Universal Robots PolyScope program: TEST_SUB_109.urp

Program TEST_SUB_109 (installation=GD directory=/programs/GD createdIn=5.13.0 lastSavedIn=5.13.0 robotSerialNumber=20235201009)
Calibrated DH parameters: a=[0.000068, -0.459527, -0.565386, -0.00004, -0.000074, 0]; d=[0.180653, 1135.485256, -1146.280412, 10.969393, 0.119732, 0.115458]; alpha=[1.570272, -0.000356, 0.007489, 1.569439, -1.570428, 0]; deltaTheta=[0, -0.72179, 6.862965, 0.14202, 0, 0]
InitVariablesNode
BeforeStart
  Script file /programs/GD/ROVI/ROVI_RESET.script
    | def ROVI_RESET():
    |   if (not socket_open(host,port,socket_name)):
    |     rovi_err=902
    |     return False
    |   end
    |   socket_send_line("X0()",socket_name)
    |   ret=socket_read_line(socket_name,socket_timeout)
    |   if (ret == "OK"):
    |     rovi_err=0
    |   elif (ret == "NG"):
    |     rovi_err=to_num(socket_read_line(socket_name,socket_timeout))
    |   else:
    |     ret="NG"
    |     rovi_err=903
    |   end
    |   socket_close(socket_name)
    |   if (rovi_err != 0):
    |     if (is_popup):
    |       popup(str_cat(ret,rovi_err),title="X0",warning=True,blocking=True)
    |     end
    |     return False
    |   else:
    |     return True
    |   end
    | end
  Script file /programs/GD/ROVI/ROVI_CAPTURE.script
    | def ROVI_CAPTURE():
    |   Y1=[0.0,0.0,0.0,0.0]
    | #  p=get_actual_tool_flange_pose()
    |   p=Bucket
    |   if (not socket_open(host,port,socket_name)):
    |     rovi_err=902
    |     return False
    |   end
    |   socket_send_string("X1(",socket_name)
    |   socket_send_string(p[0],socket_name)
    |   socket_send_string(",",socket_name)
    |   socket_send_string(p[1],socket_name)
    |   socket_send_string(",",socket_name)
    |   socket_send_string(p[2],socket_name)
    |   socket_send_string(",",socket_name)
    |   socket_send_string(p[3],socket_name)
    |   socket_send_string(",",socket_name)
    |   socket_send_string(p[4],socket_name)
    |   socket_send_string(",",socket_name)
    |   socket_send_string(p[5],socket_name)
    |   socket_send_line(")",socket_name)
    |   ret=socket_read_line(socket_name,socket_timeout)
    |   if (ret == "OK"):
    |     rovi_err=0
    |     f=socket_read_ascii_float(4,socket_name,socket_timeout)
    |     while (f[0]!=4):
    |       sleep(0.3)
    |       f=socket_read_ascii_float(4,socket_name,socket_timeout)
    |     end
    |     i=0
    |     while (i<4):
    |       Y1[i]=f[i+1]
    |       i=i+1
    |     end
    |   elif (ret == "NG"):
    |     rovi_err=to_num(socket_read_line(socket_name,socket_timeout))
    |   else:
    |     ret="NG"
    |     rovi_err=903
    |   end
    |   socket_close(socket_name)
    |   if (rovi_err != 0):
    |     if (is_popup):
    |       popup(str_cat(ret,rovi_err),title="X1",warning=True,blocking=True)
    |     end
    |     return False
    |   else:
    |     return True
    |   end
    | end
  Script file /programs/GD/ROVI/ROVI_SOLVE.script
    | def ROVI_SOLVE(is_popup=is_popup):
    |   buf=p[10000.0,0.0,0.0,0.0,0.0,0.0]
    |   if (not socket_open(host,port,socket_name)):
    |     rovi_err=902
    |     return False
    |   end
    |   socket_send_line("X2()",socket_name)
    |   ret=socket_read_line(socket_name,socket_timeout)
    |   if (ret == "OK"):
    |     rovi_err=0
    |     f=socket_read_ascii_float(6,socket_name,socket_timeout)
    |     while (f[0]!=6):
    |       sleep(0.3)
    |       f=socket_read_ascii_float(6,socket_name,socket_timeout)
    |     end
    |     counter=0
    |     while (counter<6):
    |       buf[counter]=f[counter+1]
    |       counter=counter+1
    |     end
    |   elif (ret == "NG"):
    |     rovi_err=to_num(socket_read_line(socket_name,socket_timeout))
    |   else:
    |     ret="NG"
    |     rovi_err=903
    |   end
    |   sleep(1.0)
    |   socket_close(socket_name)
    |   if (rovi_err != 0):
    |     if (is_popup):
    |       popup(str_cat(ret,rovi_err),title="X2",warning=True,blocking=True)
    |     end
    |   end
    |   return buf
    | end
  Script file /programs/GD/ROVI/ROVI_RECIPE.script
    | def ROVI_RECIPE(recipe):
    |   if (not socket_open(host,port,socket_name)):
    |     rovi_err=902
    |     return False
    |   end
    |   socket_send_line(str_cat(str_cat("X3(",recipe),")"),socket_name)
    |   ret=socket_read_line(socket_name,socket_timeout)
    |   if (ret == "OK"):
    |     rovi_err=0
    |   elif (ret == "NG"):
    |     rovi_err=to_num(socket_read_line(socket_name,socket_timeout))
    |   else:
    |     ret="NG"
    |     rovi_err=903
    |   end
    |   socket_close(socket_name)
    |   if (rovi_err != 0):
    |     if (is_popup):
    |       popup(str_cat(ret,rovi_err),title="X3",warning=True,blocking=True)
    |     end
    |     return False
    |   else:
    |     return True
    |   end
    | end
  Script file /programs/GD/ROVI/ROVI_PARAM.script
    | def ROVI_PARAM(prm_name,prm_value=None):
    |   Y8=0.0
    |   if (not socket_open(host,port,socket_name)):
    |     rovi_err=902
    |     return False
    |   end
    |   socket_send_string("X8(",socket_name)
    |   socket_send_string(prm_name,socket_name)
    |   if (prm_value != None):
    |     socket_send_string(" ",socket_name)
    |     socket_send_string(prm_value,socket_name)
    |   end
    |   socket_send_line(")",socket_name)
    |   ret=socket_read_line(socket_name,socket_timeout)
    |   if (ret == "OK"):
    |     rovi_err=0
    |     if (prm_value == None):  # rosparam get
    |       Y8=to_num(socket_read_line(socket_name,socket_timeout))
    |     else:    # rosparam set
    |       f=1
    |     end
    |   elif (ret == "NG"):
    |     rovi_err=to_num(socket_read_line(socket_name,socket_timeout))
    |   else:
    |     ret="NG"
    |     rovi_err=903
    |   end
    |   socket_close(socket_name)
    |   if (rovi_err != 0):
    |     if (is_popup):
    |       popup(str_cat(ret,rovi_err),title="X8",warning=True,blocking=True)
    |     end
    |     return False
    |   else:
    |     return True
    |   end
    | end
  Script file /programs/GD/CONTROL/CYCLE_CONTROL.script
    | def GET_REG(prg_no):
    |   WorkPosNo=read_input_integer_register(4)-1                       # GPII_WorkPosNo
    |   CaptIndex[WorkPosNo]=read_input_integer_register(21)-1           # GPII_CaptColNo
    |   CaptRowNo=read_input_integer_register(20)-1        # GPII_CaptRowNo
    |   CaptStepZ=read_input_integer_register(6) / 1000.0         # GPII_CaptStepZ
    |   ReCaptNo=0
    |   if (prg_no==1203):
    |     ReCaptNo=read_input_integer_register(22)                # GPII_ReCaptNo
    |   end
    |   ReCaptZ=read_input_integer_register(7) / 1000.0         # GPII_ReCaptZ
    |   CutOffZDef=read_input_integer_register(11) / 1000.0          # GPII_CutOffZ
    |   CrankDepthFull=read_input_integer_register(10) / 1000.0   # GPII_FullDepth
    | end
    | 
    | def POSE_SUB(p, teach_frame):
    |   return pose_trans(inv(teach_frame), p)
    | end
    | 
    | def GET_BUCKET_UPPER(pos=0):
    |   if UseNewCaptPos:
    |     p=POSE_SUB(CaptPoint_C, BucketM)
    |     pX=[BKWidth/2,CaptPointL_dX,BKWidth-CaptPointR_dX]
    |     p[0]=pX[pos]
    |   else:
    |     captpos=[CaptPoint_C,CaptPoint_L,CaptPoint_R]
    |     p=captpos[pos]
    |     p=POSE_SUB(p, BucketM)
    |   end
    |   return p
    | end
    | 
    | def SET_BUCKET_DEF():
    |   BucketM=pBucketM
    |   if (WorkPosNo<0):
    |     Bucket=pBucketC
    |   else:
    |     Bucket=pBucket[WorkPosNo]
    |   end
    | end
    | 
    | def SET_BUCKET():
    |   SET_BUCKET_DEF()
    |   Bucket[2]=Bucket[2]-CaptStepZ*CaptRowNo
    | end
    | 
    | def SET_CV():
    |   CV=pCV
    | end
    | 
    | def SET_CAPT_INDEX():
    |   CaptIndexWk=CaptIndex[WorkPosNo]
    |   ReCaptZWk=0
    |   if (prg_no==1203):
    |     if   (ReCaptNo==0):
    |       if (CaptIndexWk==0):
    |         if (0<=DistPillarBak):
    |           CaptIndexWk=1
    |         else:
    |           CaptIndexWk=2
    |         end
    |         ReCaptZWk=0
    |       else:
    |         CaptIndexWk=0
    |         ReCaptZWk=0
    |       end
    |     elif (ReCaptNo==1):
    |       if (CaptIndexWk==0):
    |         CaptIndexWk=0
    |         ReCaptZWk=-ReCaptZ
    |       else:
    |         CaptIndexWk=CaptIndexWk
    |         ReCaptZWk=-ReCaptZ
    |       end
    |     else:
    |       if (CaptIndexWk==0):
    |         CaptIndexWk=0
    |         ReCaptZWk=ReCaptZ
    |       else:
    |         CaptIndexWk=CaptIndexWk
    |         ReCaptZWk=ReCaptZ
    |       end
    |     end
    |   end
    | end
    | 
    | def GET_CAPTPOS():
    |   SET_BUCKET()
    |   SET_CAPT_INDEX()
    |   if UseNewCaptPos:
    |     p=GET_BUCKET_UPPER(CaptIndexWk)
    |     p[2]=p[2]-ReCaptZWk
    |   else:
    |     captpos=[CaptPoint_C,CaptPoint_L,CaptPoint_R]
    |     p=captpos[CaptIndexWk]
    |     p[2]=p[2]-ReCaptZWk
    |     p=POSE_SUB(p, BucketM)
    |   end
    |   return p
    | end
    | 
    | def CHECK_CAPTPOS():
    |   isOK=((CaptStepZ*(read_input_integer_register(20)-1)) < (read_input_integer_register(9) / 1000.0))
    |   return isOK
    | end
    | 
    | def GET_ZSLIDE_POS(p):
    |   p[2]=p[2]-CaptStepZ*CaptRowNo
    |   return p
    | end
    | 
    | def END_CYCLE():
    |   stopl(1.2)
    |   end_force_mode()
    |   end_freedrive_mode()
    |   socket_close(socket_name)
    | end
    | 
    | def CHECK_SPEED(smax,f=[1,1,1,1,1,1]):
    |   s=TCPSpeed
    |   i=0
    |   while (i<6):
    |     if ((f[i]==1) and (smax[i]<s[i])):
    |       return False
    |     end
    |     i=i+1
    |   end
    |   return True
    | end
  Script file /programs/GD/CONTROL/ROTATE_CONTROL.script
    | def GET_TCP_FORCE_TOOL():
    |   force_torque=get_tcp_force()
    |   force_B=p[force_torque[0], force_torque[1], force_torque[2], 0, 0, 0]
    |   torque_B=p[force_torque[3], force_torque[4], force_torque[5], 0, 0, 0]
    |   tcp=get_actual_tcp_pose()
    |   rotation_BT=p[0, 0, 0, tcp[3], tcp[4], tcp[5]]
    |   force_T=pose_trans(pose_inv(rotation_BT), force_B)
    |   torque_T=pose_trans(pose_inv(rotation_BT), torque_B)
    |   force_torque_T=p[force_T[0], force_T[1], force_T[2], torque_T[0], torque_T[1], torque_T[2]]
    |   return force_torque_T
    | end
    | 
    | def CHECK_VALUE_RZ():
    |   return True
    | end
    | 
    | def GET_FORCE_VALUE_RZ(target):
    |   PoseSub= pose_sub (CurrPos_p,target)
    |   RYSub=r2d(PoseSub[4])
    |   RZSub=r2d(PoseSub[5])
    | #  if (RYSub<RZSupRYRange[0] or RZSupRYRange[1]<RYSub):
    | #    RZSupForceVal=0.0
    | #    return RZSupForceVal
    | #  end
    |   if (RZSub<0):
    |     RZMin=RZSupDegMin[0]
    |     RZRatio=RZSupRatio[0]
    |     RZOffset=RZSupOffset[0]
    |   else:
    |     RZMin=RZSupDegMin[1]
    |     RZRatio=RZSupRatio[1]
    |     RZOffset=-RZSupOffset[1]
    |   end
    |   if (norm(RZSub) >= norm(RZMin)):
    |     RZSupForceVal=(RZMin-RZSub)*RZRatio+RZOffset
    |   else:
    |     RZSupForceVal=0
    |   end
    |   if (RZSupForceVal<RZSupForceRange[0]):
    |     RZSupForceVal=RZSupForceRange[0]
    |   elif (RZSupForceRange[1]<RZSupForceVal):
    |     RZSupForceVal=RZSupForceRange[1]
    |   end
    |   if (RYSub<RZSupRYRange[0] or RZSupRYRange[1]<RYSub):
    |     RZSupForceVal=0
    |   end
    |   if ((not UseRZSupStep1) and (ForceStep==1)):
    |     RZSupForceVal=0
    |   end
    |   return RZSupForceVal
    | end
    | 
    | def GET_CVCORR_VALUE(target):
    |   PoseSub=pose_sub(CurrPos_p,target)
    |   RYSub=r2d(PoseSub[4])
    |   CVCorrRYSub=RYSub
    |   if (RYSub<0):
    |     RYMin=-CVCorrDegMin[0]
    |     RZRatio=CVCorrRatio[0]
    |     RZOffset=-CVCorrOffset[0]
    |   else:
    |     RYMin=-CVCorrDegMin[1]
    |     RZRatio=CVCorrRatio[1]
    |     RZOffset=CVCorrOffset[1]
    |   end
    |   if (norm(RYSub) >= norm(RYMin)):
    |     t=get_tcp_offset()
    |     CVCorrYVal=-t[2]*sin(d2r(RYSub))
    |     CVCorrRZVal=RYSub*RZRatio+RZOffset
    |   else:
    |     CVCorrYVal=0
    |     CVCorrRZVal=0
    |   end
    | end
    | 
    | def GET_CVCORR_POS(target):
    |   if UseCVCorr:
    |     pos= pose_add (p[0,0,0,0,0,d2r(-CVCorrRZVal)],p[0,0,0,target[3],target[4],target[5]])
    |     pos=p[target[0],target[1],target[2],pos[3],pos[4],pos[5]]
    |   else:
    |     pos=target
    |   end
    |   return pos
    | end
  Script file /programs/GD/CONTROL/ZONE_CONTROL.script
    | def GET_DIST(P1, P2):
    |   return pose_dist(P1, P2)
    | end
    | def CHECK_DIST_NEAR(P1, P2, th):
    |   return (GET_DIST(P1, P2) < th)
    | end
    | def DIST_HOME():
    |   return pose_dist(gHome_Position,CurrPos_p)
    | end
    | 
    | def CHECK_HOME():
    |   return (DIST_HOME()<ZoneDistTh)
    | end
    | 
    | def DIST_CVFront():
    |   if (read_input_integer_register(4)==1):
    |     p=g2GD_pos1
    |   else:
    |     p=g1GD_pos1
    |   end
    |   return pose_dist(p,CurrPos_p)
    | end
    | 
    | def CHECK_CVFront():
    |   return (DIST_CVFront()<ZoneDistTh)
    | end
    | 
    | def CHECK_RB_POS(prg_no):
    |   ret=True
    |   if (prg_no==1001):
    |     ret=CHECK_ALLOW_GO_HOME(0)
    |   end
    |   if ((prg_no==1201) or (prg_no==1401) or (prg_no==1402) or (prg_no==6001) or (prg_no==6101) or (prg_no==6401) or (prg_no==6102) or (prg_no==7001)):
    |     ret=CHECK_HOME()
    |   end
    |   if ((prg_no==1002) or (prg_no==1241) or (prg_no==1261)):
    |     ret=CHECK_BKInside()
    |   end
    |   if (prg_no==1251):
    |     ret=(CHECK_HOME() or CHECK_CVUpper())
    |   end
    |   if (ret != True):
    |     SubPrgResult=801
    |     sleep(999999.0)
    |   end
    | end
    | 
    | def DIST_ORIGIN():
    |   p=CurrPos_p
    |   o=p
    |   o[0]=0.0
    |   o[1]=0.0
    |   DistOrigin=pose_dist(o,p)
    |   return pose_dist(o,p)
    | end
    | 
    | def CHECK_EVAC_ORG():
    |   return (EvacRadiusTh<DIST_ORIGIN())
    | end
    | 
    | def CHECK_EVAC_X():
    |   return (EvacXTh[0]<CurrPos_p[0] and CurrPos_p[0]<EvacXTh[1])
    | end
    | 
    | def CHECK_EVAC_Y():
    |   return (EvacYTh[0]<CurrPos_p[1] and CurrPos_p[1]<EvacYTh[1])
    | end
    | 
    | def CHECK_EVAC_Z():
    |   return (EvacZTh[0]<CurrPos_p[2] and CurrPos_p[2]<EvacZTh[1])
    | end
    | 
    | def CHECK_EVAC():
    |   ret=True
    |   ret=(ret and CHECK_EVAC_ORG())
    |   ret=(ret and CHECK_EVAC_X())
    |   ret=(ret and CHECK_EVAC_Y())
    |   ret=(ret and CHECK_EVAC_Z())
    |   return ret
    | end
    | 
    | def CHECK_BKInside():
    |   ret=True
    |   pos=read_input_integer_register(4)
    |   if (pos>2):
    |     ret=False
    |   else:
    |     if (not read_input_boolean_register(13+pos)):
    |       ret=False
    |       ver_3=read_input_boolean_register(13+pos)
    |     else:
    |       bk=pBucket[pos-1]
    |       if (pos==1):
    |         ret=(ret and CurrPos_p[0]>ZoneHomeX)
    |         ret=(ret and bk[1]-(BucketWidth-ZoneBucketGap)<CurrPos_p[1] and CurrPos_p[1]<bk[1]-ZoneBucketGap)
    |       elif (pos==2):
    |         ret=(ret and CurrPos_p[0]<-ZoneHomeX)
    |         ret=(ret and bk[1]+ZoneBucketGap<CurrPos_p[1] and CurrPos_p[1]<bk[1]+(BucketWidth-ZoneBucketGap))
    |       end
    |     end
    |   end
    |   return ret
    | end
    | 
    | def CHECK_CVOutside():
    |   ret=True
    |   ret=(ret and gCV_11_M[0]-Zone6ThX<CurrPos_p[0])
    |   ret=(ret and CurrPos_p[0]<gCV_11_M[0]+Zone6ThX)
    |   ret=(ret and gCV_11_M[1]-Zone6ThY<CurrPos_p[1])
    |   ret=(ret and CurrPos_p[1]<gCV_11_M[1]+Zone6ThY)
    |   return (not ret)
    | end
    | 
    | def CHECK_CVUpper():
    |   ret=True
    |   ret=(ret and (CVXTh[0]<CurrPos_p[0] and CurrPos_p[0]<CVXTh[1]))
    |   ret=(ret and (CVYTh[0]<CurrPos_p[1] and CurrPos_p[1]<CVYTh[1]))
    |   ret=(ret and (CVZTh[0]<CurrPos_p[2] and CurrPos_p[2]<CVZTh[1]))
    |   return ret
    | end
    | 
    | def CHECK_ALLOW_GO_HOME(no=0):
    |   ret=False
    |   if (no==0 or no==1):
    |     ret=(ret or CHECK_EVAC())
    |     v1=ret
    |   end
    |   if (no==0 or no==2):
    |     ret=(ret or CHECK_BKInside())
    |     v2=ret
    |   end
    |   if (no==0 or no==3):
    |     ret=(ret or CHECK_CVUpper())
    |     v3=ret
    |   end
    |   return ret
    | end
    | 
    | def CHECK_ZONE(no):
    |   if (no==1):
    |     return (CurrPos_p[2]>=Zone1ZTh)
    |   elif (no==2):
    |     return (CurrPos_p[0]>ZoneHomeX)
    |   elif (no==3):
    |     return (CurrPos_p[0]<-ZoneHomeX)
    |   elif (no==4):
    |     return CHECK_CVFront()
    |   elif (no==5):
    |     return CHECK_BKInside()
    |   elif (no==6):
    |     return CHECK_CVOutside()
    |   elif (no==7):
    |     return CHECK_CVUpper()
    |   end
    | end
Robot Program (runOnlyOnce=true)
  prg_no := 1201
  Set NoAction tcp=TCP_RXF
  SetPayload (workpieceName=k2)
  Folder ROVI_RECIPE
    If (not ROVI_RECIPE(GPII_WorkNo+WorkNoTL))
      SubPrgResult := rovi_err
      Wait Sleep waitTime=999999
  Folder ROVI_RESET
    If (not ROVI_RESET())
      SubPrgResult := rovi_err
      Wait Sleep waitTime=999999
  Folder ROVI_CAPTURE
    Set SingleDigitalPulseActionState SingleDigitalPulseActionState(hiPulseInSeconds=1, pin=GP_bool_out[14])
    Script: force_mode_set_damping(0)
    Script: force_mode_set_gain_scaling(0.5)
    Wait Sleep waitTime=0.02
    Script: zero_ftsensor()
    Force Frame feature=Joint_6_name; selection=[0, 0, 0, 1, 0, 0]; wrench=[0, 30, 0, 5, 10, 0]; limitsForce=[0.15, 0.03, 0.01, 0.087266, 0.087266, 1.047198]; limitsMotion=[0.1, 0.1, 0.1, 0.349066, 0.349066, 0.349066]
      var_2 := True
      SuppressedNode
        If var_2
          If TCPForce[3]>4 (checkContinuously=true)
            Wait Sleep waitTime=1
            var_2 := False
          Wait Sleep waitTime=3
      Loop While (checkContinuously=false) expression=var_2
        If TCPForce[3]<-2 (checkContinuously=true)
          Wait Sleep waitTime=1
          var_2 := False
        Wait Sleep waitTime=0.1
    Wait Sleep waitTime=3
    Script: force_mode_set_gain_scaling(1)
    Script: force_mode_set_damping(0)
    If ( not ROVI_CAPTURE())
      SubPrgResult := rovi_err
      Wait Sleep waitTime=999999
  Folder ROVI_SOLVE
    Y2 := ROVI_SOLVE()
    If (Y2[0]≟10000.)
      SubPrgResult := rovi_err
      Wait Sleep waitTime=999999
  SetPayload (workpieceName=k10)
  UF := Y2
  MoveL speed 200 mm/s, acceleration 70 mm/s^2 (useActiveTCP=false) tcp=TCP_1; feature=UF
    Wait Sleep waitTime=1
    Waypoint Variable (Variable): variable(featureName=gCV_11_M)
    Waypoint Variable (Variable): variable(featureName=gCV_12_M)
  MoveL speed 200 mm/s, acceleration 70 mm/s^2 (useActiveTCP=false) tcp=TCP_1; feature=UF
    Waypoint Variable (Variable): motionParameters(jointSpeed=1.047198 jointAcceleration=1.396263 cartesianSpeed=0.03 cartesianAcceleration=0.03); variable(featureName=gCV_13_M)
  Set SingleDigitalPulseActionState SingleDigitalPulseActionState(hiPulseInSeconds=1, pin=GP_bool_out[15])
  SuppressedNode
    Wait Sleep waitTime=3
  Halt
Thread スレッド_1 (runOnlyOnce=false)
  TCPSpeed := get_actual_tcp_speed()
  TCPForce := GET_TCP_FORCE_TOOL()
  Script: sync()
